(* CoDeSys 2.3 export: PROC_ERR_PARAMETERS.EXP *)

(* POU 60_Error handling/Process Errors/proc_Err_Parameters, ST *)
PROGRAM proc_Err_Parameters
VAR
END_VAR
;
END_PROGRAM
